// TIA Portal V17 export
// export: Created 2023-06-23T18:33:39.3415189Z, ExportSetting WithDefaults, DisplayName Totally Integrated Automation Portal, DisplayVersion V17, DisplayName TIA Portal Openness, DisplayVersion V17, DisplayName TIA Portal Version Control Interface, DisplayVersion V17, DisplayName STEP 7 Professional, DisplayVersion V17, DisplayName STEP 7 Safety, DisplayVersion V17, DisplayName WinCC Advanced / Unified PC, DisplayVersion V17
VAR_GLOBAL   // PLC tag table "16_AE2-SA1"
   "iAE2-SA1p" AT %I9.2 : Bool;   // 6
   "iAE2-SA1" AT %I9.3 : Bool;   // 6
   "iAE2-SA1a" AT %I17.3 : Bool;
   "oAE2-SA1p" AT %Q8.5 : Bool;
   "oAE2-SA1" AT %Q8.6 : Bool;
END_VAR
